TYPE STATUS_IST_POS EXTENDS RobotSollPose :
STRUCT
	i_OnlineCheck : INT;
	i_CurrentStation : INT;
	i_TargetStation : INT;
END_STRUCT
END_TYPE

(* stored: Version 1.1.0.1, ProductVersion 3.1.4024.11
   DUT STATUS_IST_POS: Id {9096263d-fb6d-4732-af28-00cb16635977} *)
